(* CODESYS project dispensador_piezas.project
   CustomField01_name: CustomField01
   CustomField08_name: CustomField08
   CustomField06_name: CustomField06
   Title: ATV_IMC_Template
   CustomField09_name: CustomField09
   CustomField07_name: CustomField07
   CustomField05_name: CustomField05
   Author: Laia Sala Perez
   CustomField02_name: CustomField02
   Description: This template can be used for a correct interface with the local drive. the MANDATORY_AT_EACH_CYCLE program must be called like it is done in this application.
   CustomField04_name: CustomField04
   CustomField10_name: CustomField10
   Version: 0.0.0.0
   Company: Schneider Electric
   CustomField03_name: CustomField03

Project tree, tasks and I/O mapping:
  MyController : TM241CE24R, Schneider Electric, order no. TM241CE24R, version 4.0.3.8
    application Application
      task MAST (cyclic, interval 20 ms, priority 15, watchdog 100 ms x 1) calls principal
      function HiddenPOU [ST]
      global variables GVL
      program principal [LD]
      function block saca_cilindro [LD]
      visualisation simulacion
    DI : Digital Inputs, Schneider Electric, version 4.0.3.8
        input  iwDI_IW0 : WORD  // IW0
        input  Application.sensor_cilindro : BOOL  // IW0.I0
        input  Application.sensor_almacen : BOOL  // IW0.I1
        input  ibDI_IB1 : BYTE  // IB1
    DQ : Digital Outputs, Schneider Electric, version 4.0.3.8
        output qwDQ_QW0 : WORD  // QW0
        output qbDQ_QB1 : BYTE  // QB1
    Counters : Counters, Schneider Electric, version 4.0.3.8
    Pulse_Generators : Pulse Generators, Schneider Electric, version 4.0.3.8
    Cartridge_1 : Cartridge, Schneider Electric, version 4.0.3.8
    IO_Bus : IO bus - TM3, Schneider Electric, version 4.0.3.8
      Module_1 : TM3DQ8R/G, Schneider Electric, order no. TM3DQ8R/G, version 1.0.1.3
          output Application.recojido : BOOL  // QB0.Q0
          output Application.extendido : BOOL  // QB0.Q1
          output Application.motor : BOOL  // QB0.Q6
          unmapped channels: QB0
    COM_Bus : COM bus, Schneider Electric, version 4.0.3.8
    Ethernet_1 : Ethernet Network, Schneider Electric, version 4.0.3.8
    Serial_Line_1 : Serial line, Schneider Electric, version 4.0.3.8
      SoMachine_Network_Manager : SoMachine-Network Manager, Schneider Electric, version 4.0.0.2
    Serial_Line_2 : Serial line, Schneider Electric, version 4.0.3.8
      Modbus_Manager : Modbus Manager, Schneider Electric, version 4.0.0.2
  text list GlobalTextList
*)

// MyController/Application/GVL
VAR_GLOBAL
	marcha: BOOL;
	confirmar: BOOL;
	motor: BOOL;
	paro: BOOL;
	sensor_cilindro: BOOL;
	sensor_almacen: BOOL;
	extendido: BOOL;
	recojido: BOOL;
	piezas: WORD;
END_VAR

// MyController/Application/principal
PROGRAM principal
VAR
	etapa1: BOOL;
	etapa2: BOOL;
	etapa0: BOOL;
	saca_cil: saca_cilindro;
END_VAR
VAR // added by the converter: edge detectors and wires of the graphical bodies
    _w1, _w2, _w3 : BOOL;
END_VAR

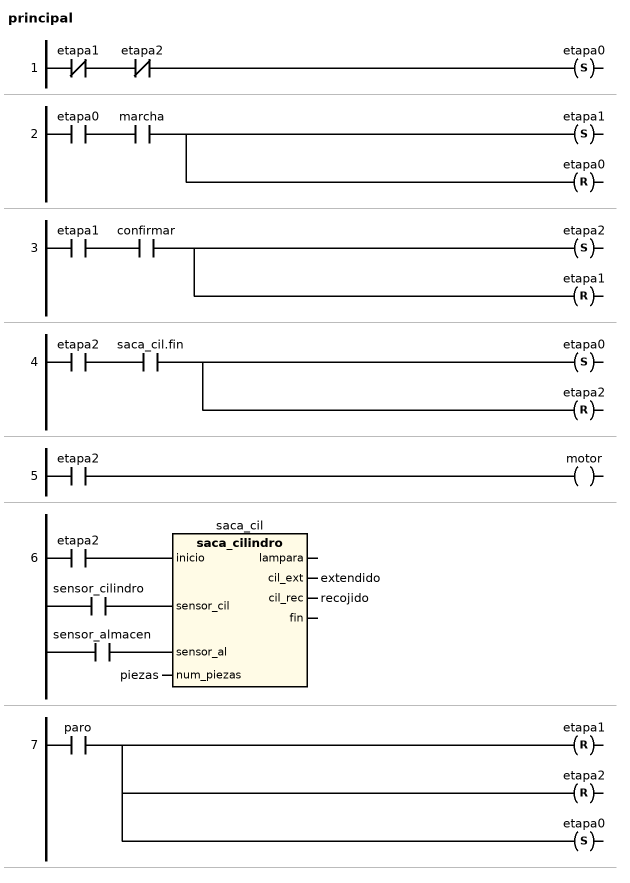
// NETWORK 1
etapa0 S= NOT etapa1 AND NOT etapa2;

// NETWORK 2
_w1 := etapa0 AND marcha;
etapa1 S= _w1;
etapa0 R= _w1;

// NETWORK 3
_w2 := etapa1 AND confirmar;
etapa2 S= _w2;
etapa1 R= _w2;

// NETWORK 4
_w3 := etapa2 AND saca_cil.fin;
etapa0 S= _w3;
etapa2 R= _w3;

// NETWORK 5
motor := etapa2;

// NETWORK 6
saca_cil(
    inicio := etapa2,
    sensor_cil := sensor_cilindro,
    sensor_al := sensor_almacen,
    num_piezas := piezas,
    cil_ext => extendido,
    cil_rec => recojido); // saca_cilindro

// NETWORK 7
etapa1 R= paro;
etapa2 R= paro;
etapa0 S= paro;

END_PROGRAM

// MyController/Application/saca_cilindro
FUNCTION_BLOCK saca_cilindro
VAR_INPUT
	inicio: BOOL;
	sensor_cil: BOOL;
	sensor_al: BOOL;
	num_piezas: WORD;
END_VAR
VAR_OUTPUT
	lampara: BOOL;
	cil_ext: BOOL;
	cil_rec: BOOL;
	fin: BOOL;
END_VAR
VAR
	etapa1: BOOL;
	etapa2: BOOL;
	etapa3: BOOL;
	etapa4: BOOL;
	etapa0: BOOL;
	temp: TON;
	cont: CTU;
	cont_reset: BOOL;
	parpadeo: BLINK;
END_VAR
VAR // added by the converter: edge detectors and wires of the graphical bodies
    _w1, _w2, _w3, _w4, _w5, _w6 : BOOL;
END_VAR

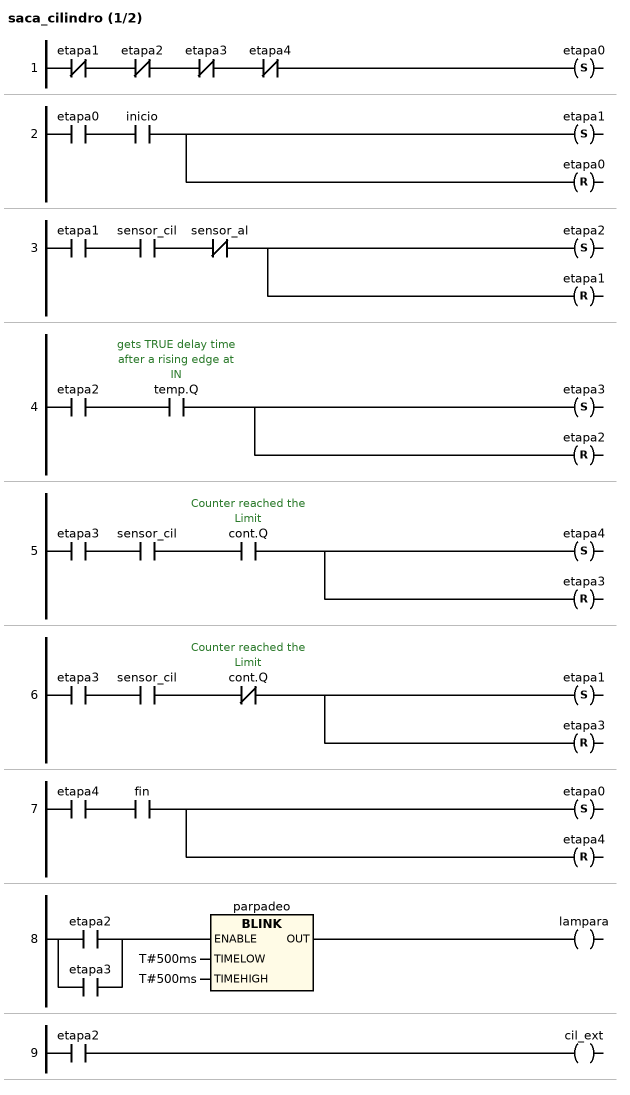
// NETWORK 1
etapa0 S= NOT etapa1 AND NOT etapa2 AND NOT etapa3 AND NOT etapa4;

// NETWORK 2
_w1 := etapa0 AND inicio;
etapa1 S= _w1;
etapa0 R= _w1;

// NETWORK 3
_w2 := etapa1 AND sensor_cil AND NOT sensor_al;
etapa2 S= _w2;
etapa1 R= _w2;

// NETWORK 4
//   temp.Q: gets TRUE delay time after a rising edge at IN
_w3 := etapa2 AND temp.Q;
etapa3 S= _w3;
etapa2 R= _w3;

// NETWORK 5
//   cont.Q: Counter reached the Limit
_w4 := etapa3 AND sensor_cil AND cont.Q;
etapa4 S= _w4;
etapa3 R= _w4;

// NETWORK 6
//   cont.Q: Counter reached the Limit
_w5 := etapa3 AND sensor_cil AND NOT cont.Q;
etapa1 S= _w5;
etapa3 R= _w5;

// NETWORK 7
_w6 := etapa4 AND fin;
etapa0 S= _w6;
etapa4 R= _w6;

// NETWORK 8
parpadeo(ENABLE := etapa2 OR etapa3, TIMELOW := T#500ms, TIMEHIGH := T#500ms); // BLINK
lampara := parpadeo.OUT;

// NETWORK 9
cil_ext := etapa2;

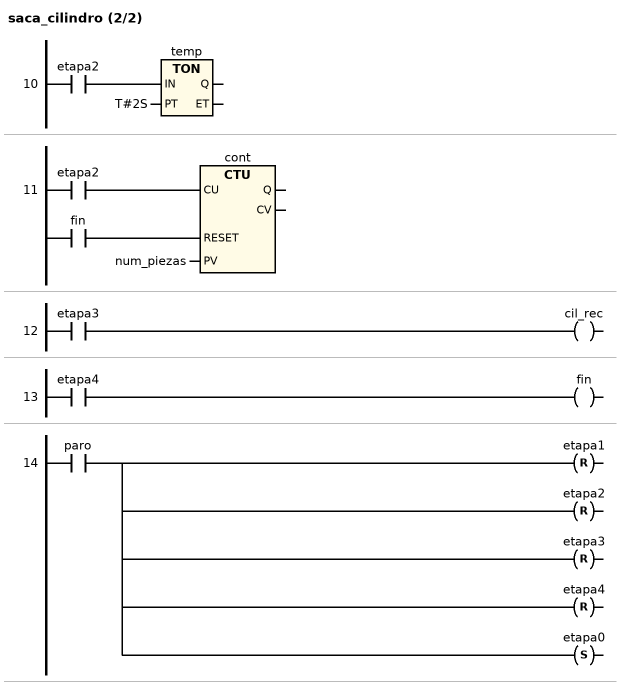
// NETWORK 10
temp(IN := etapa2, PT := T#2S); // TON

// NETWORK 11
cont(CU := etapa2, RESET := fin, PV := num_piezas); // CTU

// NETWORK 12
cil_rec := etapa3;

// NETWORK 13
fin := etapa4;

// NETWORK 14
etapa1 R= paro;
etapa2 R= paro;
etapa3 R= paro;
etapa4 R= paro;
etapa0 S= paro;

END_FUNCTION_BLOCK

// MyController/Application/HiddenPOU
FUNCTION HiddenPOU : BOOL

VAR_INPUT
	pHiddenFunc: POINTER TO WORD;
END_VAR
VAR
	pRead: POINTER TO BYTE;
	pWrite: POINTER TO BYTE;
END_VAR

pRead := pHiddenFunc + 400;
pWrite := pHiddenFunc + 4400;
HiddenPOU := TRUE;

END_FUNCTION

// MyController/Application/simulacion
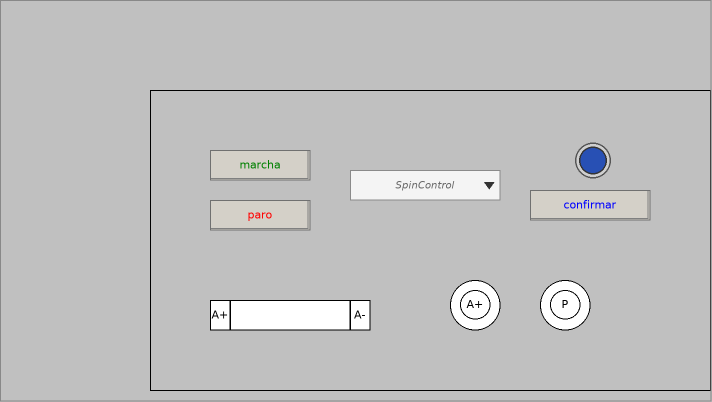
VISUALIZATION simulacion  // 712x402
    Button (210,150 100x30), "marcha"
        tap marcha
    Button (210,200 100x30), "paro"
        tap paro
    SpinControl (350,170 150x30), variable: piezas
    Button (530,190 120x30), "confirmar"
        tap confirmar
    Rectangle (230,300 120x30)
    Rectangle (350,300 20x30), "A-", colour toggle: recojido
    Rectangle (210,300 20x30), "A+", colour toggle: extendido
    Ellipse (450,280 50x50)
    Ellipse (460,290 30x29), "A+", colour toggle: sensor_cilindro
    Ellipse (540,280 50x50)
    Ellipse (550,290 30x29), "P", colour toggle: sensor_almacen
    Lamp1 (570,140 46x41), variable: principal.saca_cil.lampara, style: Lamp-Lamp1-Blue
    Line (150,100)
    Line (150,90) (710,90)
    Line (430,90) (430,90)
    Line (710,90) (710,390)
    Line (150,90) (150,390)
    Line (150,400)
    Line (150,390) (710,390)
END_VISUALIZATION
